// TwinCAT 3 PLC project RoutinePLC
// ProgramVersion: 3.1.4024.0
// libraries:
//   Tc2_Standard, * (Beckhoff Automation GmbH)
//   Tc2_System, * (Beckhoff Automation GmbH)
//   Tc3_Module, * (Beckhoff Automation GmbH)
// project tree:
//   / GlobalTextList.TcGTLO, PlcTask.TcTTO, Visualization Manager.TcVMO (not stored)
//   GVLs/ GVL.TcGVL
//   POUs/ Printing.TcPOU, PrintingStates.TcDUT, RunningStates.TcDUT, Running2.TcPOU, Visualization.TcVIS
// real-time tasks:
//   TASK PlcTask: cycle T#10ms, priority 20, ADS port 350

CONFIGURATION RoutinePLC
    RESOURCE PLC ON TwinCAT3
        TASK PlcTask(INTERVAL := T#10ms, PRIORITY := 20);
        PROGRAM Printing WITH PlcTask : Printing;
        PROGRAM Running2 WITH PlcTask : Running2;
    END_RESOURCE
END_CONFIGURATION

// ---- POUs/PrintingStates.TcDUT
TYPE PrintingStates :
(	
	PrepareModel,
	SlicePrint,
	Print,
	FinishPrint
	) := PrepareModel;
END_TYPE

// ---- POUs/RunningStates.TcDUT
TYPE RunningStates :
(	
	Start,
	Preparation,
	WarmUp,
	Running,
	EndRun
	) := Start;
END_TYPE

// ---- GVLs/GVL.TcGVL
{attribute 'qualified_only'}
VAR_GLOBAL
	RunState : RunningStates := runningstates.Start;
	PrintState : PrintingStates := printingstates.PrepareModel;
	CheckPrint : BOOL := FALSE;
	Layer1Good : BOOL := FALSE;
	Layer1Bad : Bool := False;
	EntryPrint:BOOL:=TRUE;
	PrintStarted: BOOL := FALSE;
	PrintFinished: BOOL := FALSE;
END_VAR

// ---- POUs/Printing.TcPOU
PROGRAM Printing
VAR
	CadModel: BOOL;
	StlFile: BOOL;
	Preheat: BOOL;
	EntrySlice: BOOL;
	PrintSettings: BOOL;
	Slice: BOOL;
	TransferFile: BOOL;
	PreheatTimer :TON;
	EntryPrint: BOOL;
	StartPrint: BOOL;
	Checkprint1: BOOL;
	ContinuePrint: BOOL;
	PrintComplete: BOOL;
	FinishPrintEntry: BOOL;
	RemovePrint: BOOL;
	CleanBed: BOOL;
	PrintSucceeded: BOOL;
	PrintFinished: BOOL;
	PrintFailed:BOOL;
	PrintStatePrepareModel: BOOL;
	PrintStateSlicePrint: BOOL;
	PrintStatePrint: BOOL;
	PrintStateFinishPrint: BOOL;
END_VAR


CASE gvl.PrintState OF

//Prepare state for modeling and converting 3d-print	
PrintingStates.PrepareModel:
PrintStatePrepareModel:=TRUE;
PrintStateSlicePrint:=FALSE;
PrintStatePrint:=FALSE;
PrintStateFinishPrint:=FALSE;

IF gvl.EntryPrint = TRUE THEN
	gvl.EntryPrint := FALSE;
	CadModel := TRUE;
END_IF
IF Cadmodel = TRUE THEN
	StlFile :=TRUE;
	Cadmodel:=FALSE;
END_IF
IF StlFile = TRUE THEN
	Preheat :=TRUE;
	StlFile:=FALSE;
END_IF
IF Preheat = TRUE THEN
	gvl.PrintState := printingstates.SlicePrint;
	Preheat := FALSE;
	EntrySlice :=TRUE;
END_IF

//Second State, Slice the print
PrintingStates.SlicePrint:
PrintStatePrepareModel:=FALSE;
PrintStateSlicePrint:=TRUE;
PrintStatePrint:=FALSE;
PrintStateFinishPrint:=FALSE;

PreheatTimer(in:=TRUE,PT:=T#10S); //preheat printer
IF EntrySlice = TRUE THEN
	EntrySlice:=FALSE;
	PrintSettings:=TRUE;	
END_IF
IF PrintSettings THEN
	PrintSettings:= FALSE;
	Slice :=TRUE;
END_IF
IF Slice THEN
	Slice :=FALSE;
	TransferFile:=TRUE;
END_IF
IF Transferfile = TRUE AND PreheatTimer.Q = TRUE THEN
	TransferFile:=FALSE;
	GVL.PrintState :=PrintingStates.Print;
	EntryPrint:=TRUE;
END_IF

//Third state of printing
PrintingStates.Print:
PrintStatePrepareModel:=FALSE;
PrintStateSlicePrint:=FALSE;
PrintStatePrint:=TRUE;
PrintStateFinishPrint:=FALSE;

IF EntryPrint THEN
	Entryprint :=FALSE;	
	StartPrint := TRUE;
END_IF
IF Startprint THEN
	Startprint := FALSE;
	Checkprint1 := TRUE;
	gvl.PrintStarted:=TRUE; //Signal to start Running routine
END_IF

IF Checkprint1 THEN 
	IF gvl.Layer1Good = TRUE THEN //If the first layer is good, continue proces and start running proces
		Checkprint1:=FALSE;			//Button in visualization to make true
		ContinuePrint := TRUE;
		
	ELSIF gvl.Layer1Bad = TRUE THEN
	checkprint1 := FALSE;
	GVL.PrintState := printingstates.SlicePrint; //If the first layer failed, go back to the slicing settings	
	END_IF
END_IF
IF ContinuePrint THEN
	ContinuePrint:=FALSE;
	PrintComplete:= TRUE;
END_IF
IF PrintComplete THEN
	GVL.PrintState:=PrintingStates.FinishPrint;
	PrintComplete:=FALSE;
	FinishPrintEntry:=TRUE;
END_IF

//Last state of printing proces
PrintingStates.FinishPrint:
PrintStatePrepareModel:=FALSE;
PrintStateSlicePrint:=FALSE;
PrintStatePrint:=FALSE;
PrintStateFinishPrint:=TRUE;
IF FinishPrintEntry THEN
	FinishPrintEntry:=FALSE;
	RemovePrint:=TRUE;
END_IF
IF Removeprint THEN
	Removeprint:=FALSE;
	CleanBed:=TRUE;
END_IF
IF CleanBed THEN
	IF PrintSucceeded THEN //Button in visualization to make true
		PrintFinished:=TRUE;
		CleanBed:=FALSE;
	ELSIF PrintFailed THEN
		gvl.PrintState:=PrintingStates.SlicePrint;
		CleanBed:=FALSE;
		EntrySlice:= TRUE;
	END_IF
END_IF
IF printFinished THEN
	gvl.PrintFinished:=TRUE;
	PrintFinished:=FALSE;
	gvl.Printstate:=PrintingStates.PrepareModel;
END_IF

END_CASE

END_PROGRAM

// ---- POUs/Running2.TcPOU
PROGRAM Running2
VAR
	entryR1:BOOL:=FALSE;	
	CheckWeather: BOOL;
	WeatherClear: BOOL := TRUE;
	Timer1 : TON ;
	RunTime:TON;
	CooldownTime:TON;
	ChangeClothes: BOOL;
	WatchOn: BOOL;
	EarbudsConnected: BOOL;
	MusicPlaying: BOOL;
	SearchGps: BOOL;
	EntryR2: BOOL;
	RunningShoesOn: BOOL;
	Timer2: TON;
	Outside: BOOL;
	Timer1_2: TON;
	GPSConnected: BOOL;
	WarmUp:BOOL;
	Timer2_2: TON;
	EntryRunning: BOOL;
	Running:BOOL;
	PrepFinished: BOOL;
	EntryWarmUp: BOOL;
	CheckDistance: INT;
	RunFinished: BOOL;
	EndRunEntry: BOOL;
	Cooldown: BOOL;
	GoHome: BOOL;
	Rest: BOOL;
	DrinkWater: BOOL;
	Shower: BOOL;
	RunstateStart: BOOL;
	RunstatePreperation: BOOL;
	RunstateWarmup: BOOL;
	RunstateRunning: BOOL;
	RunstateEndRun: BOOL;
END_VAR

CASE gvl.RunState OF 
Runningstates.Start:
RunstateStart:=TRUE;
RunstatePreperation:=FALSE;
RunstateWarmup:=FALSE;
RunstateRunning:=FALSE;
RunstateEndRun:=FALSE;

IF gvl.PrintStarted THEN //Check for the printer to have started in printing routine
	gvl.PrintStarted:=FALSE;
	EntryR1:=TRUE;
	gvl.RunState:=Runningstates.Preparation;
END_IF

//First State of running
Runningstates.Preparation:
RunstateStart:=FALSE;
RunstatePreperation:=TRUE;
RunstateWarmup:=FALSE;
RunstateRunning:=FALSE;
RunstateEndRun:=FALSE;
Timer1(in:=TRUE,pt:=T#2S);
Timer1_2(in:=TRUE,pt:=T#10S);

IF EntryR1 = TRUE THEN
CheckWeather := TRUE;
EntryR1 := FALSE;
END_IF


IF CheckWeather = TRUE AND WeatherClear = TRUE THEN //Use button in visualization to set WeatherClear
CheckWeather := FALSE;
ChangeClothes := TRUE;
WatchOn:= TRUE;
EarbudsConnected :=TRUE;
MusicPlaying := TRUE;
END_IF

IF Changeclothes = TRUE AND WatchOn= TRUE AND EarbudsConnected =TRUE AND MusicPlaying = TRUE AND Timer1.Q = TRUE THEN
ChangeClothes := FALSE;
WatchOn:= FALSE;    
EarbudsConnected :=FALSE;
MusicPlaying := FALSE;
Timer1.in :=FALSE;
PrepFinished :=TRUE;
END_IF

//First check print in second program before continuïng
IF gvl.Layer1Good = TRUE AND PrepFinished =TRUE THEN
SearchGps := TRUE;
EntryR2 := TRUE;
PrepFinished:=FALSE;	
END_IF

IF SearchGPS = TRUE AND EntryR2 = TRUE THEN
EntryR2 := FALSE;
RunningShoesOn:= TRUE;	
END_IF

IF RunningShoesOn = TRUE AND Timer1_2.Q THEN
gvl.RunState := RunningStates.Warmup;	
Timer1_2(in:=FALSE);
EntryWarmUp:=TRUE;
END_IF

//Second State of running
RunningStates.WarmUp:
RunstateStart:=FALSE;
RunstatePreperation:=FALSE;
RunstateWarmup:=TRUE;
RunstateRunning:=FALSE;
RunstateEndRun:=FALSE;
Timer2(In:=TRUE,PT:=T#5M);

IF EntryWarmUp THEN
Outside := TRUE;	
END_IF

IF Outside =TRUE AND GPSConnected = TRUE THEN //Button in visualization for gpsconnected
WarmUp:=TRUE;
Timer2_2(in:=TRUE,PT:=T#5S);//5 minutes warm-up, set to seconds for time-purpose
END_IF

IF timer2_2.Q = TRUE AND warmup THEN
	gvl.RunState := Runningstates.Running;
	EntryRunning:=TRUE;
	Timer2_2(in:=FALSE);
	Warmup:=FALSE;
END_IF

//Third State of running, the actual run
Runningstates.Running:
RunstateStart:=FALSE;
RunstatePreperation:=FALSE;
RunstateWarmup:=FALSE;
RunstateRunning:=TRUE;
RunstateEndRun:=FALSE;
Runtime(IN:=TRUE,pt:=T#50M);
IF EntryRunning = TRUE THEN
	Running := TRUE;
	entryRunning:=FALSE;
END_IF
IF Running AND Runtime.ET = T#50S THEN //Used time instead of distance for this program
RunFinished:=TRUE;
Runtime.IN:=TRUE;
END_IF
IF Runfinished THEN
	RunFinished:=FALSE;
	gvl.RunState:=Runningstates.EndRun;
	EndRunEntry:=TRUE;
END_IF

Runningstates.EndRun:
RunstateStart:=FALSE;
RunstatePreperation:=FALSE;
RunstateWarmup:=FALSE;
RunstateRunning:=FALSE;
RunstateEndRun:=TRUE;
IF EndRunEntry THEN	
Cooldown:= TRUE;
CoolDownTime(in:=TRUE,pt:=T#5M);
END_IF
IF Cooldown AND cooldowntime.Q THEN
	Cooldowntime.IN:=FALSE;
	Cooldown:=FALSE;
	EndrunEntry:=FALSE;
	GoHome:=TRUE;
END_IF
IF GoHome THEN
	GoHome:=FALSE;
	Rest:=TRUE;
	RunningShoesOn:=FALSE;
END_IF
IF Rest=TRUE AND RunningShoesOn = FALSE THEN
	Rest:=FALSE;
	DrinkWater:=TRUE;
	
END_IF
IF DrinkWater AND gvl.PrintFinished THEN
	Shower :=TRUE;
	Drinkwater :=FALSE;
	gvl.PrintFinished:=FALSE;
END_IF
IF Shower THEN
	shower:=FALSE;
	gvl.RunState:=RunningStates.Start;
END_IF
END_CASE

END_PROGRAM

// ---- GlobalTextList.TcGTLO
TEXTLIST GlobalTextList
  911 = 'Active Printing State'
  167 = 'End Run'
  890 = 'Finish'
  833 = 'Finish Print'
  858 = 'GPS Connected'
  175 = 'Layer 1 Bad'
  387 = 'Layer 1 Good'
  887 = 'Prep Model'
  799 = 'Prepare Model'
  435 = 'Preperation'
  659 = 'Print'
  285 = 'Print Buttons And States'
  9 = 'Print Failed'
  506 = 'Print Reset'
  609 = 'Print Start'
  509 = 'Print Succeeded'
  54 = 'Printing.PrintStateText'
  622 = 'Run Buttons And States'
  10 = 'Running'
  983 = 'Slice'
  640 = 'Slice Print'
  789 = 'Start'
  92 = 'Warm up'
  957 = 'Weather Clear'
END_TEXTLIST

// ---- POUs/Visualization.TcVIS
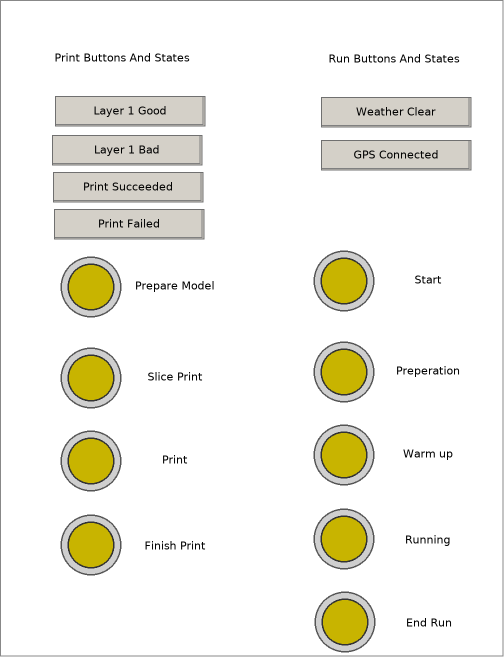
VISUALIZATION Visualization  // 504x657
    Button (321,97 150x30), "Weather Clear"
        tap Running2.WeatherClear
    Button (321,140 150x30), "GPS Connected"
        tap Running2.GPSConnected
    Button (55,96 150x30), "Layer 1 Good"
        tap GVL.Layer1Good
    Button (52,135 150x30), "Layer 1 Bad"
        tap GVL.Layer1Bad
    Lamp1 (56,252 70x70), variable: Printing.PrintStatePrepareModel, style: Lamp-Lamp1-Yellow
    Lamp1 (56,343 70x70), variable: Printing.PrintStateSlicePrint, style: Lamp-Lamp1-Yellow
    Lamp1 (56,426 70x70), variable: Printing.PrintStatePrint, style: Lamp-Lamp1-Yellow
    Lamp1 (56,510 70x70), variable: Printing.PrintStateFinishPrint, style: Lamp-Lamp1-Yellow
    Button (53,172 150x30), "Print Succeeded"
        tap Printing.PrintSucceeded
    Button (54,209 150x30), "Print Failed"
        tap GVL.Layer1Good
    Label (47,43 150x30), "Print Buttons And States"
    Label (100,271 150x30), "Prepare Model"
    Label (100,362 150x30), "Slice Print"
    Label (100,445 150x30), "Print"
    Label (100,531 150x30), "Finish Print"
    Label (319,44 150x30), "Run Buttons And States"
    Lamp1 (309,246 70x70), variable: Running2.RunstateStart, style: Lamp-Lamp1-Yellow
    Lamp1 (309,337 70x70), variable: Running2.RunstatePreperation, style: Lamp-Lamp1-Yellow
    Lamp1 (309,420 70x70), variable: Running2.RunstateWarmup, style: Lamp-Lamp1-Yellow
    Lamp1 (309,504 70x70), variable: Running2.RunstateRunning, style: Lamp-Lamp1-Yellow
    Label (353,265 150x30), "Start"
    Label (353,356 150x30), "Preperation"
    Label (353,439 150x30), "Warm up"
    Label (353,525 150x30), "Running"
    Lamp1 (310,587 70x70), variable: Running2.RunstateEndRun, style: Lamp-Lamp1-Yellow
    Label (354,608 150x30), "End Run"
END_VISUALIZATION
